// TIA Portal V17 export
// export: Created 2024-09-27T18:53:46.4196643Z, ExportSetting WithDefaults, DisplayName Totally Integrated Automation Portal, DisplayVersion V17, DisplayName TIA Portal Openness, DisplayVersion V17, DisplayName TIA Portal Version Control Interface, DisplayVersion V17, DisplayName STEP 7 Professional, DisplayVersion V17, DisplayName STEP 7 Safety, DisplayVersion V17, DisplayName WinCC Professional, DisplayVersion V17
FUNCTION "SERVO" : Void   // FC4, LAD
{ S7_Optimized_Access := 'TRUE' }
VERSION : 0.1
// stored: AutoNumber true, IsIECCheckEnabled false, SetENOAutomatically false, UDAEnableTagReadback false
   VAR_TEMP
      Actual_position : Real;
   END_VAR
   VAR_TEMP   // added for the SCL form of the ladder/FBD networks
      _w1 : Bool;
   END_VAR
BEGIN

REGION Network 1: POWER ON
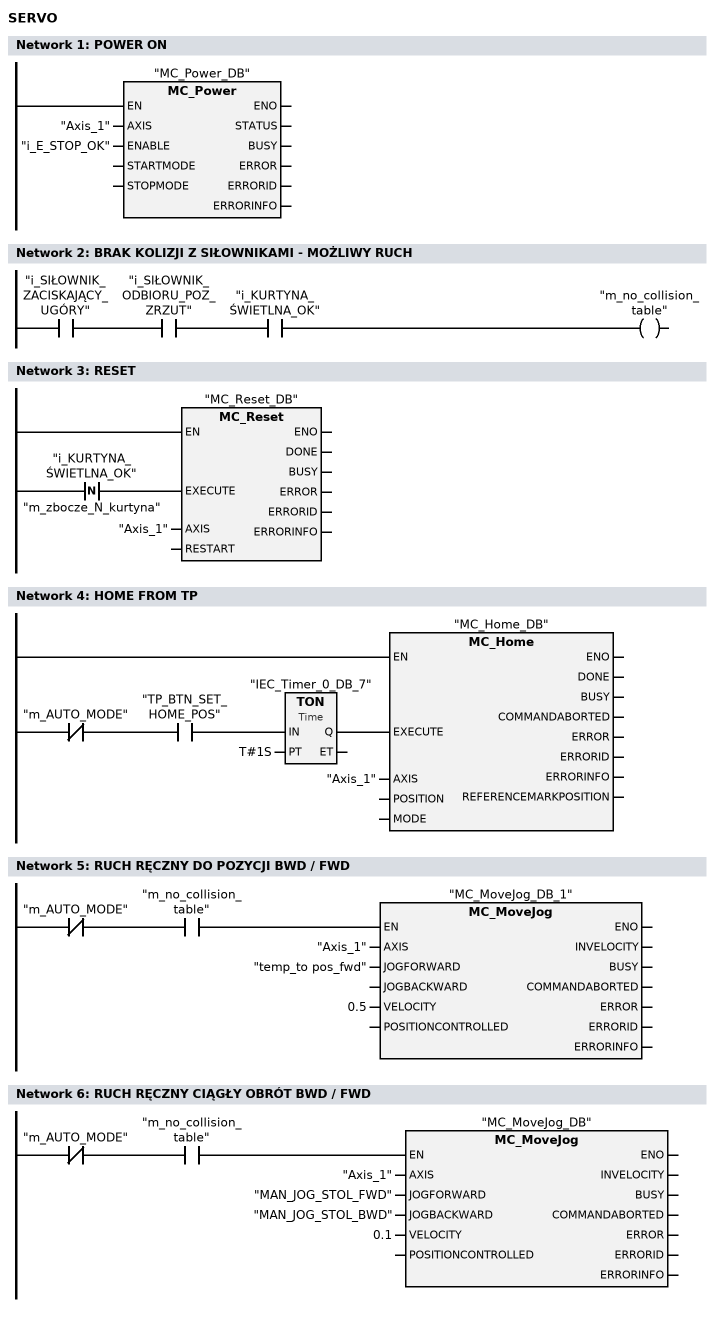
   RUNG wire#powerrail
      "MC_Power_DB".MC_Power(Axis := "Axis_1", Enable := "i_E_STOP_OK", StartMode :=, StopMode :=, Status =>, Busy =>, Error =>, ErrorID =>, ErrorInfo =>)
   END_RUNG
   // the same network as SCL:
   "MC_Power_DB"(Axis := "Axis_1", Enable := "i_E_STOP_OK");   // MC_Power
END_REGION

REGION Network 2: BRAK KOLIZJI Z SIŁOWNIKAMI - MOŻLIWY RUCH
   RUNG wire#powerrail
      Contact( "i_SIŁOWNIK_ZACISKAJĄCY_UGÓRY" )
      Contact( "i_SIŁOWNIK_ODBIORU_POZ_ZRZUT" )
      Contact( "i_KURTYNA_ŚWIETLNA_OK" )
      Coil( "m_no_collision_table" )
   END_RUNG
   // the same network as SCL:
   "m_no_collision_table" := "i_SIŁOWNIK_ZACISKAJĄCY_UGÓRY" AND "i_SIŁOWNIK_ODBIORU_POZ_ZRZUT" AND "i_KURTYNA_ŚWIETLNA_OK";
END_REGION

REGION Network 3: RESET
   RUNG wire#powerrail
      "MC_Reset_DB".MC_Reset(Execute := wire#w1, Axis := "Axis_1", Restart :=, Done =>, Busy =>, Error =>, ErrorID =>, ErrorInfo =>)
   END_RUNG
   RUNG wire#powerrail
      N_Contact(operand := "i_KURTYNA_ŚWIETLNA_OK", bit := "m_zbocze_N_kurtyna")
   END_RUNG wire#w1
   // the same network as SCL:
   #_w1 := NOT "i_KURTYNA_ŚWIETLNA_OK" AND "m_zbocze_N_kurtyna";   // falling edge of "i_KURTYNA_ŚWIETLNA_OK"
   "m_zbocze_N_kurtyna" := "i_KURTYNA_ŚWIETLNA_OK";
   "MC_Reset_DB"(Execute := #_w1, Axis := "Axis_1");   // MC_Reset
END_REGION

REGION Network 4: HOME FROM TP
   RUNG wire#powerrail
      "MC_Home_DB".MC_Home(Execute := wire#w1, Axis := "Axis_1", Position :=, Mode :=, Done =>, Busy =>, CommandAborted =>, Error =>, ErrorID =>, ErrorInfo =>, ReferenceMarkPosition =>)
   END_RUNG
   RUNG wire#powerrail
      I_Contact( "m_AUTO_MODE" )
      Contact( "TP_BTN_SET_HOME_POS" )
      { S7_Templates := "time_type := Time" } "IEC_Timer_0_DB_7".TON(pt := T#1S, et =>)
   END_RUNG wire#w1
   // the same network as SCL:
   "IEC_Timer_0_DB_7".TON(IN := NOT "m_AUTO_MODE" AND "TP_BTN_SET_HOME_POS", PT := T#1S);
   "MC_Home_DB"(Execute := "IEC_Timer_0_DB_7".Q, Axis := "Axis_1");   // MC_Home
END_REGION

REGION Network 5: RUCH RĘCZNY DO POZYCJI BWD / FWD
   RUNG wire#powerrail
      I_Contact( "m_AUTO_MODE" )
      Contact( "m_no_collision_table" )
      "MC_MoveJog_DB_1".MC_MoveJog(Axis := "Axis_1", JogForward := "temp_to pos_fwd", JogBackward :=, Velocity := 0.5, PositionControlled :=, InVelocity =>, Busy =>, CommandAborted =>, Error =>, ErrorID =>, ErrorInfo =>)
   END_RUNG
   // the same network as SCL:
   IF NOT "m_AUTO_MODE" AND "m_no_collision_table" THEN
       "MC_MoveJog_DB_1"(Axis := "Axis_1", JogForward := "temp_to pos_fwd", Velocity := 0.5);   // MC_MoveJog
   END_IF;
END_REGION

REGION Network 6: RUCH RĘCZNY CIĄGŁY OBRÓT BWD / FWD
   RUNG wire#powerrail
      I_Contact( "m_AUTO_MODE" )
      Contact( "m_no_collision_table" )
      "MC_MoveJog_DB".MC_MoveJog(Axis := "Axis_1", JogForward := "MAN_JOG_STOL_FWD", JogBackward := "MAN_JOG_STOL_BWD", Velocity := 0.1, PositionControlled :=, InVelocity =>, Busy =>, CommandAborted =>, Error =>, ErrorID =>, ErrorInfo =>)
   END_RUNG
   // the same network as SCL:
   IF NOT "m_AUTO_MODE" AND "m_no_collision_table" THEN
       "MC_MoveJog_DB"(Axis := "Axis_1",   // MC_MoveJog
                       JogForward := "MAN_JOG_STOL_FWD",
                       JogBackward := "MAN_JOG_STOL_BWD",
                       Velocity := 0.1);
   END_IF;
END_REGION
END_FUNCTION
